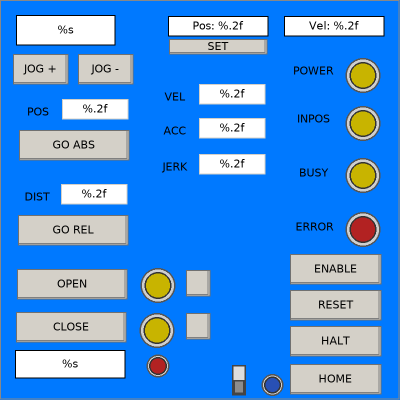
VISUALIZATION vAXIS  // 400x400
VAR_IN_OUT
	vAxis:FB_Axis;
END_VAR
    Rectangle (168,16 100x20), "Pos: %.2f", text variable: vAxis.rActPos
    Rectangle (284,16 100x20), "Vel: %.2f", text variable: vAxis.rActVel
    Lamp1 (343,53 40x45), variable: vAxis.power.Enable, style: Lamp-Lamp1-Yellow
    Label (286,60 55x22), "POWER"
    Lamp1 (343,101 40x45), variable: vAxis.bInPos, style: Lamp-Lamp1-Yellow
    Lamp1 (343,207 40x45), variable: vAxis.bAXIS_ERROR, style: Lamp-Lamp1-Red
    Lamp1 (343,153 40x45), variable: vAxis.bBusy, style: Lamp-Lamp1-Yellow
    Label (286,108 55x22), "INPOS"
    Label (287,216 55x22), "ERROR"
    Label (286,162 55x22), "BUSY"
    Button (290,254 91x30), "ENABLE"
        toggle vAxis.bEnable
    Button (290,290 91x30), "RESET"
        toggle vAxis.bReset
    Button (290,326 91x30), "HALT"
        tap vAxis.bHalt
    Textfield (199,84 66x20), "%.2f", text variable: vAxis.rVel
        OnMouseDown: write the text variable via Default
    Label (157,86 36x22), "VEL"
    Textfield (62,99 66x20), "%.2f", text variable: vAxis.rPos
        OnMouseDown: write the text variable via Default
    Label (20,101 36x22), "POS"
    Textfield (199,154 66x20), "%.2f", text variable: vAxis.rJerk
        OnMouseDown: write the text variable via Default
    Label (157,156 36x22), "JERK"
    Textfield (199,118 66x20), "%.2f", text variable: vAxis.rAcc
        OnMouseDown: write the text variable via Default
    Label (157,120 36x22), "ACC"
    Button (13,54 55x30), "JOG +"
        tap vAxis.bJogPos
    Button (78,54 55x30), "JOG -"
        tap vAxis.bJogNeg
    Button (19,130 110x30), "GO ABS"
        OnMouseDown: execute { vAXIS.bMoveABS:=TRUE; }
    Textfield (61,184 66x20), "%.2f", text variable: vAxis.Dist
        OnMouseDown: write the text variable via Default
    Label (19,186 36x22), "DIST"
    Button (18,215 110x30), "GO REL"
        OnMouseDown: execute { vAXIS.bMoveRel:=TRUE; }
    Rectangle (16,15 99x30), "%s", text variable: vAxis.sName
    Button (169,39 98x15), "SET"
        tap vAxis.bSetPosition
    Button (17,269 110x30), "OPEN"
        OnMouseDown: execute { vAXIS.bOPEN:=TRUE;  vAXIS.bCLOSE:=FALSE; }
    Button (16,312 110x30), "CLOSE"
        OnMouseDown: execute { vAXIS.bCLOSE:=TRUE; vAXIS.bOPEN:=FALSE; }
    Lamp1 (138,263 40x45), variable: vAxis.bLIMIT_OPENED, style: Lamp-Lamp1-Yellow
    Lamp1 (137,308 40x45), variable: vAxis.bLIMIT_CLOSED, style: Lamp-Lamp1-Yellow
    Rectangle (15,350 110x28), "%s", text variable: vAxis.sAXIS_STATE
    Button (186,270 24x26)
        toggle vAxis.bLIMIT_OPENED
    Button (186,313 24x26)
        toggle vAxis.bLIMIT_CLOSED
    Button (290,364 91x30), "HOME"
        OnMouseDown: execute { vAxis.bHOME:=TRUE; }
    DipSwitch (224,365 30x30), variable: vAxis.bHOME_DIR, behaviour: TOGGLE, style: Switch-DipSwitch-Gray
    Lamp1 (260,368 25x34), variable: vAxis.bHOMED, style: Lamp-Lamp1-Blue
    Lamp1 (145,352 26x28), variable: vAxis.bSTATE_ERROR;, style: Lamp-Lamp1-Red
END_VISUALIZATION

(* stored: Version 1.1.0.1, ProductVersion 3.1.4024.12
   Visu vAXIS: Id {d5d97f89-906b-489b-9dde-74bb1e2b7ed8} *)
